// TIA Portal V16 export
// export: Created 2023-03-29T11:05:04.634659Z, ExportSetting WithDefaults, DisplayName Totally Integrated Automation Portal, DisplayVersion V16 Update 6, DisplayName TIA Portal Version Control Interface, DisplayVersion V16 Update 2, DisplayName TIA Portal Openness, DisplayVersion V16 Update 6, DisplayName STEP 7 Professional, DisplayVersion V16 Update 6, DisplayName STEP 7 Safety, DisplayVersion V16, DisplayName WinCC Advanced, DisplayVersion V16 Update 6
VAR_GLOBAL   // PLC tag table "MP04_1"
   temp_current_fow_H_Q1 AT %MW600 : Word;   // H byte przepływ aktualny VF
   tmp_current_fow_L_Q1 AT %MW602 : Word;   // L byte przepływ aktualny VF
   tmp_front_volumeVF_H_Q1 AT %MW604 : Word;   // licznik objetości przód H byte
   tmp_front_volumeVF_L_Q1 AT %MW606 : Word;   // licznik objetości przód L byte
   tmp_back_balueVR_H_Q1 AT %MW608 : Word;   // licznik objętości wstecz H byte
   tmp_back_balueVR_L_Q1 AT %MW610 : Word;   // licznik objętości wstecz L byte
   "tmp_differential counter VD_H_Q1" AT %MW612 : Word;   // licznik różnicowy VD H byte
   "tmp_differential counter VD_L_Q1" AT %MW614 : Word;   // licznik różnicowy VD L byte
   "tmp_volume counter status _GF_H_Q1" AT %MW616 : Word;   // statu licznik objetości GF H byte
   "tmp_volume counter status _GF_L_Q1" AT %MW618 : Word;   // status licznik objetości GF L byte
   "tmp_volume counter status_GR_H_Q1" AT %MW620 : Word;   // statu licznik objetości GR H byte
   "tmp_volume counter status_GR_L_Q1" AT %MW622 : Word;   // statu licznik objetości GR L byte
   "tmp_differential counter status_GD_H_Q1" AT %MW624 : Word;   // statu licznik objetości GD H byte
   "tmp_differential counter status_GD_L_Q1" AT %MW626 : Word;   // statu licznik objetości GD L byte
   tmp_sataus_MP04_Q1 AT %MW628 : Word;   // staus urządzenia MP04_Q1
   temp_current_fow_H_Q2 AT %MW630 : Word;   // H byte przepływ aktualny VF
   tmp_current_fow_L_Q2 AT %MW632 : Word;   // L byte przepływ aktualny VF
   tmp_front_volumeVF_H_Q2 AT %MW634 : Word;   // licznik objetości przód H byte
   tmp_front_volumeVF_L_Q2 AT %MW636 : Word;   // licznik objetości przód L byte
   tmp_back_balueVR_H_Q2 AT %MW638 : Word;   // licznik objętości wstecz H byte
   tmp_back_balueVR_L_Q2 AT %MW640 : Word;   // licznik objętości wstecz L byte
   "tmp_differential counter VD_H_Q2" AT %MW642 : Word;   // licznik różnicowy VD H byte
   "tmp_differential counter VD_L_Q2" AT %MW644 : Word;   // licznik różnicowy VD L byte
   "tmp_volume counter status _GF_H_Q2" AT %MW646 : Word;   // statu licznik objetości GF H byte
   "tmp_volume counter status _GF_L_Q2" AT %MW648 : Word;   // status licznik objetości GF L byte
   "tmp_volume counter status_GR_H_Q2" AT %MW650 : Word;   // statu licznik objetości GR H byte
   "tmp_volume counter status_GR_L_Q2" AT %MW652 : Word;   // statu licznik objetości GR L byte
   "tmp_differential counter status_GD_H_Q2" AT %MW654 : Word;   // statu licznik objetości GD H byte
   "tmp_differential counter status_GD_L_Q2" AT %MW656 : Word;   // statu licznik objetości GD L byte
   tmp_sataus_MP04_Q2 AT %MW658 : Word;   // staus urządzenia MP04_Q2
END_VAR
